{attribute 'qualified_only'}
{attribute 'strict'}
{attribute 'to_string'}
TYPE E_States :
(
    Waiting := 0,
    HasCoin,
    ProductEjected,
    CoinEjected
);
END_TYPE

(* stored: Version 1.1.0.1, ProductVersion 3.1.4024.9
   DUT E_States: Id {dc88566f-2d51-4930-b010-ad814213063f} *)
